PROGRAM Dtank_Pivot_To_Window
VAR
    setPos : MC_SetPosition;
    nominalPosition : LREAL := 1673;
END_VAR

GVL.astAxes[AXIS_DTANK_PIVOT_TO_WINDOW].stInputs.bLimitBwd := TRUE;
GVL.astAxes[AXIS_DTANK_PIVOT_TO_WINDOW].stInputs.bLimitFwd := TRUE;
GVL.astAxes[AXIS_DTANK_PIVOT_TO_WINDOW].stControl.bEnable := TRUE;



IF _TaskInfo[fbGetCurTaskIndex.index].FirstCycle THEN
    //Initial default values:
    setPos.Execute:= TRUE;
END_IF


setPos.Position := nominalPosition;

setPos(Axis:= astAxes[AXIS_DTANK_PIVOT_TO_WINDOW].Axis);
setPos.Execute:= FALSE;

END_PROGRAM

(* stored: Version 1.1.0.1, ProductVersion 3.1.4024.11
   POU Dtank_Pivot_To_Window: Id {80308c5a-8765-4ec4-96d3-88987add8d1c}, SpecialFunc None *)
